{attribute addProperty BoxType "KL8519"}
{attribute addProperty Id "Channel_1Channel_48E8280200"}
{attribute addProperty CRC "2933714008"}
{attribute addProperty SizeInBites "0"}
{attribute addProperty SizeInBytes "0"}
TYPE KL8519_AEDCEC58 :
STRUCT
	{attribute addProperty Name "Channel_1"}
	Channel_1 : Channel_48E82802;
END_STRUCT
END_TYPE

(* stored: Version 1.2.0.0, ProductVersion 3.1.4024.9
   DUT KL8519_AEDCEC58: Id {ef195627-4235-41e3-8293-9e6700a26c99} *)
